FUNCTION_BLOCK FB_BiDirectionConveyer
VAR_INPUT
END_VAR
VAR_OUTPUT
END_VAR
VAR
END_VAR

END_FUNCTION_BLOCK

(* stored: Version 1.1.0.1, ProductVersion 3.1.4024.16
   POU FB_BiDirectionConveyer: Id {9bbb15e2-4ac3-4493-ba62-1b0aee54c0f3}, SpecialFunc None *)
